TYPE T_Ctrl_SIf_PTS_Ilk :
STRUCT
END_STRUCT
END_TYPE

(* stored: Version 1.1.0.1, ProductVersion 3.1.0.23
   DUT T_Ctrl_SIf_PTS_Ilk: Id {e1f40279-d222-40d4-8985-d3a7abb27105} *)
